FUNCTION_BLOCK CompositeFB3
  (* Standard: 61499-2 *)
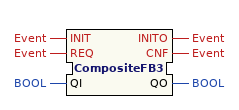
  EVENT_INPUT
    INIT;
    REQ;
  END_EVENT
  EVENT_OUTPUT
    INITO;
    CNF;
  END_EVENT
  VAR_INPUT
    QI : BOOL;
  END_VAR
  VAR_OUTPUT
    QO : BOOL;
  END_VAR
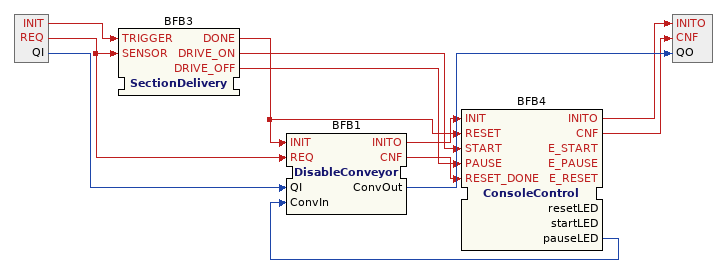
  FBS
    BFB3 : SectionDelivery;
    BFB4 : ConsoleControl;
    BFB1 : DisableConveyor;
  END_FBS
  EVENT_CONNECTIONS
    INIT TO BFB3.TRIGGER;
    REQ TO BFB3.SENSOR;
    BFB3.DONE TO BFB1.INIT;
    BFB3.DRIVE_ON TO BFB4.START;
    BFB3.DRIVE_OFF TO BFB4.PAUSE;
    BFB1.CNF TO BFB4.RESET_DONE;
    BFB1.INITO TO BFB4.INIT;
    BFB3.DONE TO BFB4.RESET;
    REQ TO BFB1.REQ;
    BFB4.CNF TO CNF;
    BFB4.INITO TO INITO;
  END_CONNECTIONS
  DATA_CONNECTIONS
    QI TO BFB1.QI;
    BFB4.pauseLED TO BFB1.ConvIn;
    BFB1.ConvOut TO QO;
  END_CONNECTIONS
END_FUNCTION_BLOCK
